PROGRAM MAIN
VAR
	Signal_IN		:	Signal_generator;
	checking		:	Signal_check;
	data_out		:	Struct_OUT;
	data_in			:	Struct_IN;
END_VAR

Signal_IN();
checking(Signal_IN:= Signal_IN.SIGNAL);
data_out.bHeat1 := checking.Signal_OUT;
data_out.bOK := checking.bOK;

END_PROGRAM

(* stored: Version 1.1.0.1, ProductVersion 3.1.4024.16
   POU MAIN: Id {05fb79fc-cb93-42b1-8606-c8378de38b2a}, SpecialFunc None *)
